// Mitsubishi GX Works2 project: 서보1   PLC: Q02/Q02H

PROGRAM MAIN
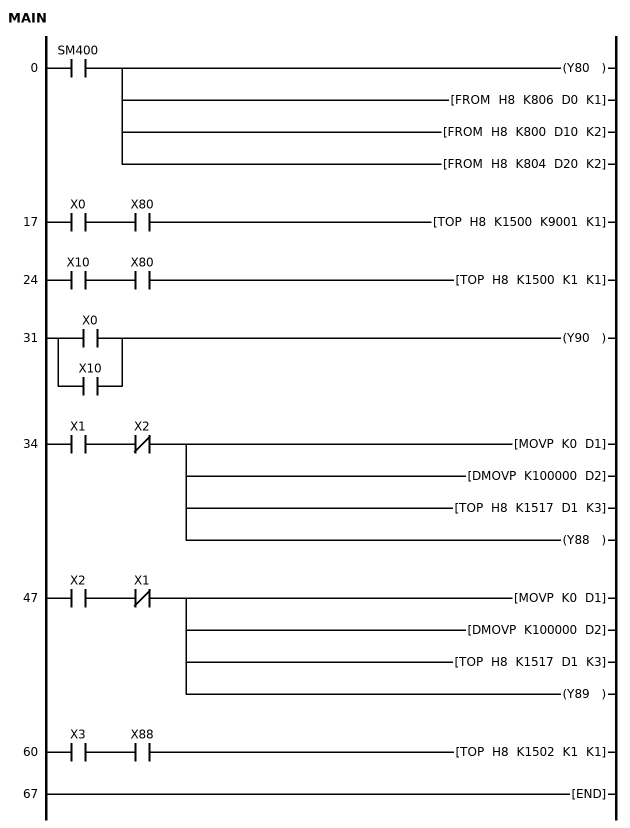
0     LD      SM400
      OUT     Y80
      FROM    H8 K806 D0 K1
      FROM    H8 K800 D10 K2
      FROM    H8 K804 D20 K2
17    LD      X0
      AND     X80
      TOP     H8 K1500 K9001 K1
24    LD      X10
      AND     X80
      TOP     H8 K1500 K1 K1
31    LD      X0
      OR      X10
      OUT     Y90
34    LD      X1
      ANI     X2
      MOVP    K0 D1
      DMOVP   K100000 D2
      TOP     H8 K1517 D1 K3
      OUT     Y88
47    LD      X2
      ANI     X1
      MOVP    K0 D1
      DMOVP   K100000 D2
      TOP     H8 K1517 D1 K3
      OUT     Y89
60    LD      X3
      AND     X88
      TOP     H8 K1502 K1 K1
67    END
END_PROGRAM
